Universal Robots PolyScope program: ATI Demo Program.urp

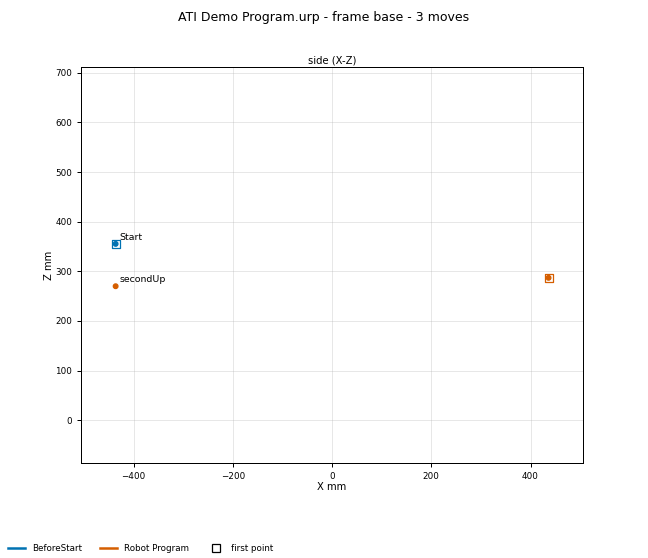
[picture p0: tool path of ATI Demo Program.urp in frame base, 3 of 9 moves have a stored position in this frame; points joined in program order, loops and branches not executed]
Program ATI Demo Program (createdIn=3.1.18024.0 lastSavedIn=3.3.0.145 directory=/home/ur/ursim-3.3.0/programs installation=default robotSerialNumber=2014359999)
Calibrated DH parameters: a=[0.000241, -0.156882, -0.391168, -0.000034, 0.000033, 0]; d=[0.08909, 1210.353649, -1202.089359, -8.154207, 0.094912, 0.082482]; alpha=[1.570962, 0.000326, -0.003342, 1.570446, -1.570439, 0]; deltaTheta=[0.000082, 1.192638, -1.263181, 0.0705, 0.00007, 0.000052]
BeforeStart
  Folder Move to Initial start position
    MoveJ speed 60 deg/s, acceleration 80 deg/s^2 (recalculateMotions=false)
      Waypoint Start: TCP in base x=-436.352 y=579.706 z=355.306 mm, rx=3.1399 ry=-0.0472 rz=-0.0056 rad; joints [-61.803, -57.175, 58.456, -91.289, 270.047, 29.954] deg
    URCap com.ur.urcap.ATI_FT.ATI FT Sensor data=running = Enable
      | WEIGHT = 0.025
Robot Program (runOnlyOnce=false motionType=MoveJ speed=1.047198 acceleration=1.396263 recalculateMotions=false)
  Folder Bias the sensor
    Wait Sleep waitTime=1
    URCap com.ur.urcap.ATI_FT.ATI FT Sensor data=running = Bias
  Folder Move down until the tool touchs a surface
    MoveL speed 40 mm/s, acceleration 200 mm/s^2 (recalculateMotions=false) feature=Base
      If force()<2 (checkContinuously=true)
        Waypoint SeekDown (Relative): relativeFromPosition TCP in base x=-99.537 y=-399.332 z=353.883 mm, rx=0.0027 ry=-3.1384 rz=-0.0008 rad; joints [-88.578, -78.615, -111.599, -79.821, 89.816, 1.322] deg; TCP in base x=-100.895 y=-399.448 z=-109.905 mm, rx=-0.0035 ry=-3.1383 rz=-0.0004 rad; joints [-88.578, -139.653, -133.528, 3.146, 89.816, 1.322] deg
  Folder Move across the surface while applying 10N of force
    Force Simple feature=Joint_6_name; selection=[0, 0, 1, 0, 0, 0]; wrench=[0, 0, 10, 0, 0, 0]; limitsForce=[0.15, 0.15, 0.15, 1.047198, 1.047198, 1.047198]; limitsMotion=[0.1, 0.1, 0.1, 0.349066, 0.349066, 0.349066]
      MoveL speed 40 mm/s, acceleration 25 mm/s^2 (recalculateMotions=false) feature=Joint_6_name
        Wait Sleep waitTime=1
        Folder If the tool encounters too much resistance, return to start position
          If xyPlaneForce < 15 (checkContinuously=true)
            Waypoint MoveForce (Relative): relativeFromPosition TCP in base x=-436.359 y=579.696 z=355.25 mm, rx=3.1399 ry=-0.0472 rz=-0.0054 rad; joints [-61.803, -57.175, 58.456, -91.289, 270.047, 29.954] deg; TCP in base x=436.38 y=579.622 z=355.372 mm, rx=3.1399 ry=-0.0472 rz=-0.0051 rad; joints [-135.73, -57.119, 58.32, -90.983, 269.918, -43.973] deg; pose in feature x=0 y=0 z=0 mm, rx=0 ry=0 rz=0 rad; flange x=436.37 y=579.672 z=355.256 mm, rx=3.1399 ry=-0.0472 rz=-0.0054 rad
  Folder Reset to a start position
    MoveL speed 250 mm/s, acceleration 1200 mm/s^2 (recalculateMotions=false) feature=Base
      Waypoint Up (Relative): relativeFromPosition TCP in base x=-436.39 y=579.651 z=262.908 mm, rx=3.1399 ry=-0.047 rz=-0.0055 rad; joints [-61.794, -55.361, 69.182, -103.829, 270.049, 29.921] deg; TCP in base x=-436.336 y=579.673 z=343.365 mm, rx=3.14 ry=-0.0472 rz=-0.0056 rad; joints [-61.802, -57.106, 60.102, -93.003, 270.047, 29.949] deg; flange x=-436.348 y=579.679 z=343.315 mm, rx=3.1399 ry=-0.0472 rz=-0.0055 rad
      Waypoint firstUp: TCP in base x=436.386 y=579.646 z=286.859 mm, rx=3.1399 ry=-0.0472 rz=-0.0054 rad; joints [-135.724, -56.056, 66.674, -100.399, 269.918, -43.997] deg
  Folder Move down until the tool touchs a surface
    MoveL speed 40 mm/s, acceleration 200 mm/s^2 (recalculateMotions=false) feature=Base
      If ForceValue<2 (checkContinuously=true)
        Waypoint SeekDown2 (Relative): relativeFromPosition TCP in base x=436.383 y=579.646 z=373.28 mm, rx=3.1399 ry=-0.0472 rz=-0.0054 rad; joints [-135.732, -57.11, 55.675, -88.345, 269.918, -43.966] deg; TCP in base x=436.373 y=579.653 z=233.631 mm, rx=3.1398 ry=-0.0472 rz=-0.0056 rad; joints [-135.719, -54.2, 71.648, -107.229, 269.922, -44.015] deg; flange x=436.37 y=579.672 z=233.681 mm, rx=3.1399 ry=-0.0472 rz=-0.0054 rad
  Folder Move across the surface while applying 10N of force
    Force Simple feature=Joint_6_name; selection=[0, 0, 1, 0, 0, 0]; wrench=[0, 0, 10, 0, 0, 0]; limitsForce=[0.15, 0.15, 0.15, 1.047198, 1.047198, 1.047198]; limitsMotion=[0.1, 0.1, 0.1, 0.349066, 0.349066, 0.349066]
      MoveL speed 40 mm/s, acceleration 25 mm/s^2 (recalculateMotions=false) feature=Joint_6_name
        Wait Sleep waitTime=1
        Folder If the tool encounters too much resistance, return to start position
          If xyPlaneForce < 15 (checkContinuously=true)
            Waypoint MoveForce2 (Relative): relativeFromPosition TCP in base x=436.341 y=579.683 z=355.309 mm, rx=3.1398 ry=-0.047 rz=-0.0053 rad; joints [-135.73, -57.119, 58.32, -90.983, 269.918, -43.973] deg; TCP in base x=-436.31 y=579.718 z=355.257 mm, rx=3.1398 ry=-0.0471 rz=-0.0053 rad; joints [-61.803, -57.175, 58.456, -91.289, 270.047, 29.954] deg; pose in feature x=0 y=0 z=0 mm, rx=0 ry=0 rz=0 rad; flange x=-436.348 y=579.679 z=355.315 mm, rx=3.1399 ry=-0.0472 rz=-0.0055 rad
  Folder Reset to a start position
    MoveL speed 150 mm/s, acceleration 400 mm/s^2 (recalculateMotions=false) feature=Base
      Waypoint Up (Relative): relativeFromPosition TCP in base x=-436.39 y=579.651 z=262.908 mm, rx=3.1399 ry=-0.047 rz=-0.0055 rad; joints [-61.794, -55.361, 69.182, -103.829, 270.049, 29.921] deg; TCP in base x=-436.336 y=579.673 z=343.365 mm, rx=3.14 ry=-0.0472 rz=-0.0056 rad; joints [-61.802, -57.106, 60.102, -93.003, 270.047, 29.949] deg; flange x=-436.348 y=579.679 z=343.315 mm, rx=3.1399 ry=-0.0472 rz=-0.0055 rad
      Waypoint secondUp: TCP in base x=-436.356 y=579.68 z=269.926 mm, rx=3.1399 ry=-0.047 rz=-0.0055 rad; joints [-61.795, -55.594, 68.513, -102.927, 270.049, 29.924] deg
Thread Thread_1 (runOnlyOnce=false trackProgramExecution=false)
  TCPForce := get_tcp_force()
  ForceValue := TCPForce[2]
  TCPPose := get_actual_tcp_pose()
  Folder Get magnitude of force in X-Y plane, accounting for friction of tool
    xyPlaneForce := sqrt(pow(TCPForce[0], 2) + pow(TCPForce[1], 2)) - 0.3*ForceValue
  Wait Sleep waitTime=0.01
